ABB RobotStudio station: 6640_station_20220131-163936.rsstn

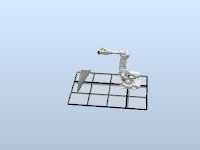
Station Station (saved by RobotStudio 21.4.9700.0)
Controller 6640_180_255
  mechanical unit ROB_1: IRB6640_180_255__04_2, 6 joints, base frame (0, 0, 0) mm
Layout (positions relative to the parent item):
  - MyNewTool [mechanism, from models\Paintgun.rslib] at (0, 0, 0) mm
  - generic_fan_blade [part, from models\generic_fan_blade.rslib] at (2700, -800, 500) mm, rotated rx 90 ry 0 rz 90 deg
  - IRB6640_180_255__04_2 [mechanism, from Robots\IRB6640_180_255_G_04.rslib] at (0, 0, 0) mm; joint values [0, 0, 0, 0, 0.5236, 0] (rad or m)
